PROGRAM MAIN
VAR
END_VAR

END_PROGRAM

(* stored: Version 1.1.0.1
   POU MAIN: Id {f84aa32f-dcff-4e09-8280-674d7af84ce0} *)
